{attribute 'GeneratedUsingTerminal: EL6080-0000-0018'}
{attribute addProperty BoxType "EL6080-0000-0018"}
{attribute addProperty Id "ControlAT %Q*UINT2"}
{attribute addProperty CRC "3674028256"}
{attribute addProperty Size "2"}
TYPE Control_DAFD38E0 :
STRUCT
	{attribute addProperty Name "Control"}
	Control AT %Q* : UINT;
END_STRUCT
END_TYPE

(* stored: Version 1.2.0.0, ProductVersion 3.1.4024.9
   DUT Control_DAFD38E0: Id {42cc9567-96b7-44c0-afb4-76b24bd490da} *)
